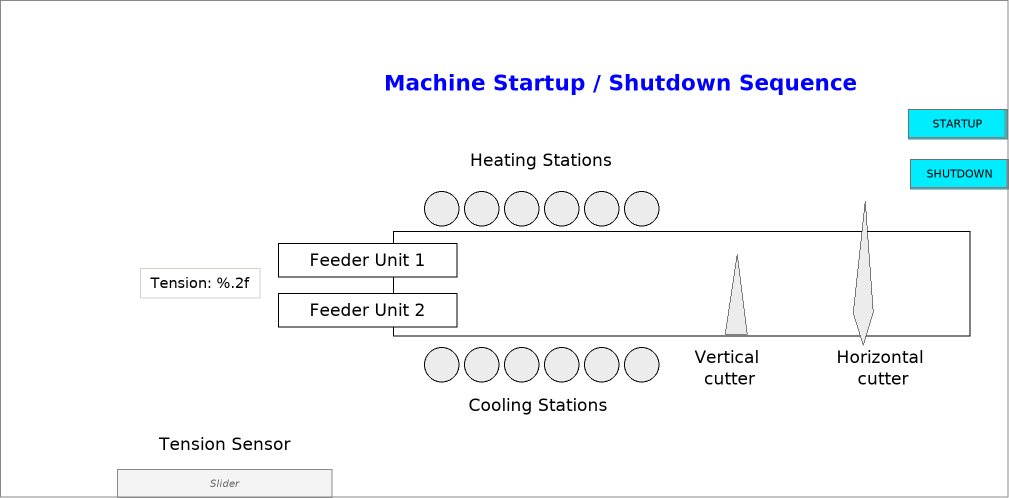
VISUALIZATION MachineStartupShutdownSequence  // 1009x498
    Rectangle (393,231 577x105)
    Ellipse (424,191 35x35), colour toggle: MAIN.MachineStartupShutdownSequence.HeatingStation[1]
    Ellipse (464,191 35x35), colour toggle: MAIN.MachineStartupShutdownSequence.HeatingStation[2]
    Ellipse (424,347 35x35), colour toggle: MAIN.MachineStartupShutdownSequence.CoolStation[1]
    Ellipse (464,347 35x35), colour toggle: MAIN.MachineStartupShutdownSequence.CoolStation[2]
    Ellipse (504,191 35x35), colour toggle: MAIN.MachineStartupShutdownSequence.HeatingStation[3]
    Ellipse (544,191 35x35), colour toggle: MAIN.MachineStartupShutdownSequence.HeatingStation[4]
    Ellipse (504,347 35x35), colour toggle: MAIN.MachineStartupShutdownSequence.CoolStation[3]
    Ellipse (544,347 35x35), colour toggle: MAIN.MachineStartupShutdownSequence.CoolStation[4]
    Rectangle (278,243 179x34), "Feeder Unit 1", colour toggle: MAIN.MachineStartupShutdownSequence.FeederUnit1
    Rectangle (278,293 179x34), "Feeder Unit 2", colour toggle: MAIN.MachineStartupShutdownSequence.FeederUnit2
    Ellipse (584,191 35x35), colour toggle: MAIN.MachineStartupShutdownSequence.HeatingStation[5]
    Ellipse (624,191 35x35), colour toggle: MAIN.MachineStartupShutdownSequence.HeatingStation[6]
    Ellipse (584,347 35x35), colour toggle: MAIN.MachineStartupShutdownSequence.CoolStation[5]
    Ellipse (624,347 35x35), colour toggle: MAIN.MachineStartupShutdownSequence.CoolStation[6]
    Slider (117,469 215x29), variable: MAIN.MachineStartupShutdownSequence.WindingTension, scale 0..20
    Button (908,109 99x30), "STARTUP", colour toggle: MAIN.MachineStartupShutdownSequence.StartupRun
        tap MAIN.SeqStart
    Textfield (140,268 120x30), "Tension: %.2f", text variable: MAIN.MachineStartupShutdownSequence.WindingTension
    Polygon (725,334) (747,334) (737,254), colour toggle: MAIN.MachineStartupShutdownSequence.VerticalCutter, invisible if: MAIN.tp02.Q AND MAIN.MachineStartupShutdownSequence.VerticalCutter
    Polygon (853,313) (863,345) (873,312) (865,201), colour toggle: MAIN.MachineStartupShutdownSequence.HorizontalCutter, invisible if: MAIN.tp04.Q AND MAIN.MachineStartupShutdownSequence.HorizontalCutter
    Label (458,145 166x30), "Heating Stations"
    Label (455,390 166x30), "Cooling Stations"
    Button (910,159 99x30), "SHUTDOWN", colour toggle: MAIN.MachineStartupShutdownSequence.ShutdownRun
        tap MAIN.SeqStop
    Label (380,68 481x30), "Machine Startup / Shutdown Sequence"
    Label (677,333 105x70), "Vertical cutter"
    Label (829,337 108x62), "Horizontal cutter"
    Label (146,424 158x40), "Tension Sensor"
END_VISUALIZATION

(* stored: Version 1.1.0.1, ProductVersion 3.1.4024.15
   Visu MachineStartupShutdownSequence: Id {e2c6e81f-0aac-4bd6-838c-daab2644b6d3} *)
